FUNCTION_BLOCK CLIENT_5_4 (* 5 SD/4 RD Client Interface *)
  (* Standard: 61499-1; Function: Communication; Description: 5SD/4RD Client *)
  (* Version 0.0, 2003-04-10, JHC, Rockwell Automation *)
  (* Compiler header: package fb.rt.net; *)
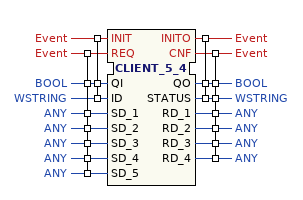
  EVENT_INPUT
    INIT WITH QI, ID;
    REQ WITH QI, SD_1, SD_2, SD_3, SD_4, SD_5;
  END_EVENT
  EVENT_OUTPUT
    INITO WITH QO, STATUS;
    CNF WITH QO, STATUS, RD_1, RD_2, RD_3, RD_4;
  END_EVENT
  VAR_INPUT
    QI : BOOL;
    ID : WSTRING;
    SD_1 : ANY;
    SD_2 : ANY;
    SD_3 : ANY;
    SD_4 : ANY;
    SD_5 : ANY;
  END_VAR
  VAR_OUTPUT
    QO : BOOL; (* Event Output Qualifier *)
    STATUS : WSTRING; (* Service Status *)
    RD_1 : ANY; (* Received Data *)
    RD_2 : ANY;
    RD_3 : ANY;
    RD_4 : ANY;
  END_VAR
END_FUNCTION_BLOCK
